Xinje XDPPro project, PLC1: XD5-60-6Pls (software 3.4 2016-10-12)

PROGRAM Ladder

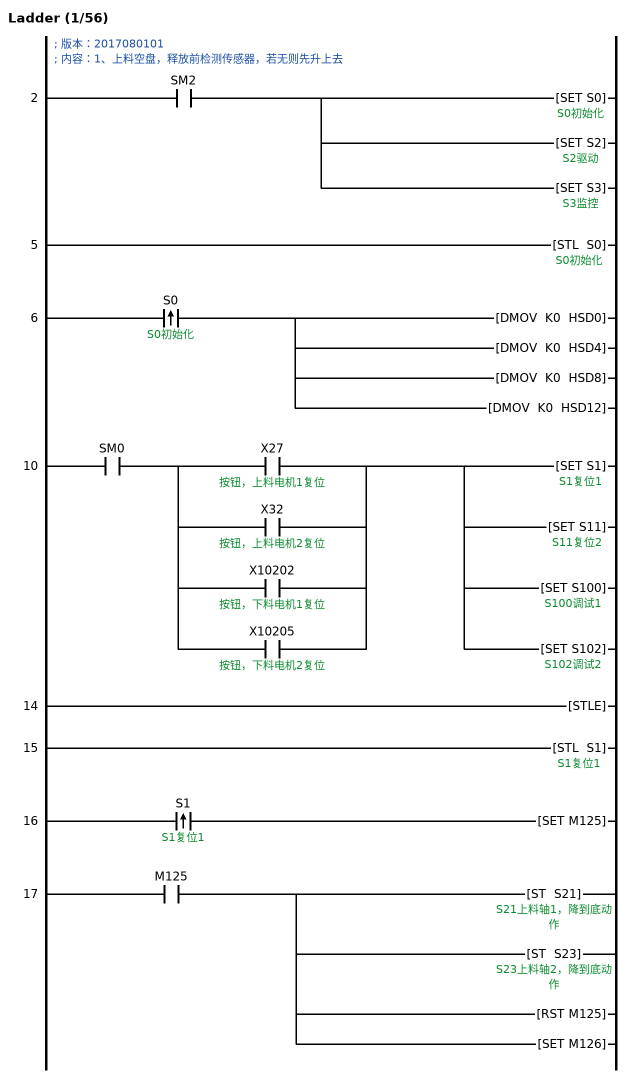
; 版本：2017080101
; 内容：1、上料空盘，释放前检测传感器，若无则先升上去
LD     SM2
SET    S0	; S0初始化
SET    S2	; S2驱动
SET    S3	; S3监控
STL    S0	; S0初始化
LDP    S0	; S0初始化
DMOV   K0 HSD0
DMOV   K0 HSD4
DMOV   K0 HSD8
DMOV   K0 HSD12
LD     SM0
LD     X27	; 按钮，上料电机1复位
OR     X32	; 按钮，上料电机2复位
OR     X10202	; 按钮，下料电机1复位
OR     X10205	; 按钮，下料电机2复位
ANB
SET    S1	; S1复位1
SET    S11	; S11复位2
SET    S100	; S100调试1
SET    S102	; S102调试2
STLE
STL    S1	; S1复位1
LDP    S1	; S1复位1
SET    M125
LD     M125
ST     S21	; S21上料轴1，降到底动作
ST     S23	; S23上料轴2，降到底动作
RST    M125
SET    M126

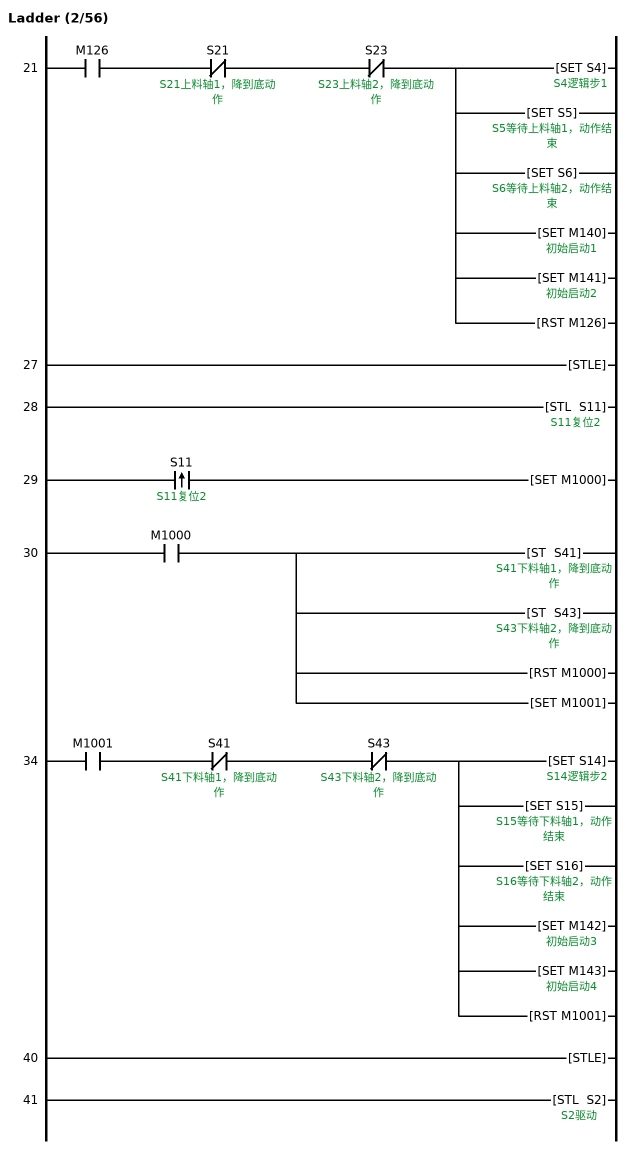
LD     M126
ANI    S21	; S21上料轴1，降到底动作
ANI    S23	; S23上料轴2，降到底动作
SET    S4	; S4逻辑步1
SET    S5	; S5等待上料轴1，动作结束
SET    S6	; S6等待上料轴2，动作结束
SET    M140	; 初始启动1
SET    M141	; 初始启动2
RST    M126
STLE
STL    S11	; S11复位2
LDP    S11	; S11复位2
SET    M1000
LD     M1000
ST     S41	; S41下料轴1，降到底动作
ST     S43	; S43下料轴2，降到底动作
RST    M1000
SET    M1001
LD     M1001
ANI    S41	; S41下料轴1，降到底动作
ANI    S43	; S43下料轴2，降到底动作
SET    S14	; S14逻辑步2
SET    S15	; S15等待下料轴1，动作结束
SET    S16	; S16等待下料轴2，动作结束
SET    M142	; 初始启动3
SET    M143	; 初始启动4
RST    M1001
STLE
STL    S2	; S2驱动

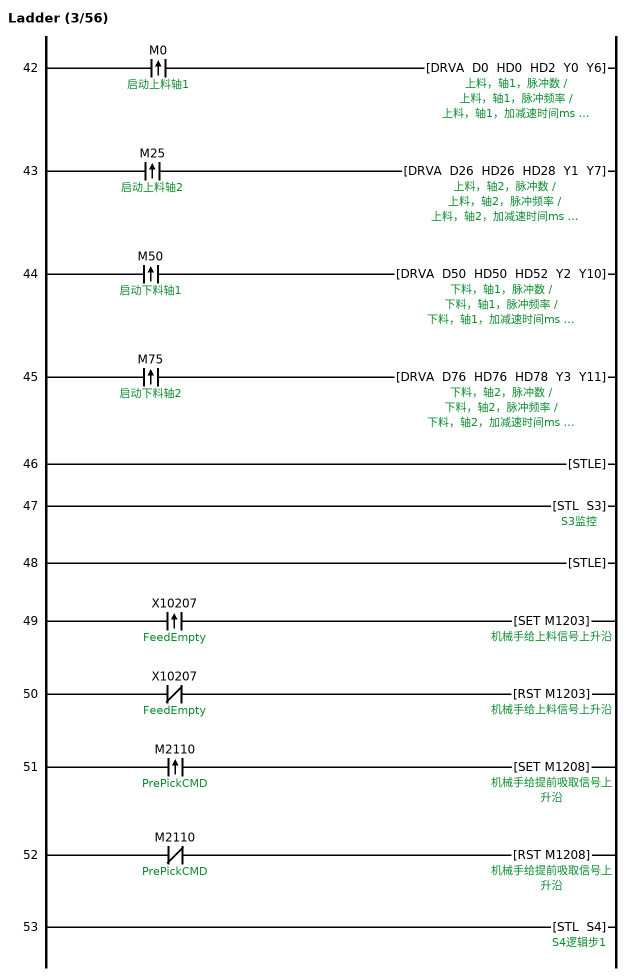
LDP    M0	; 启动上料轴1
DRVA   D0 HD0 HD2 Y0 Y6	; 上料，轴1，脉冲数 / 上料，轴1，脉冲频率 / 上料，轴1，加减速时间ms / 上料1电机脉冲 / 上料1电机方向
LDP    M25	; 启动上料轴2
DRVA   D26 HD26 HD28 Y1 Y7	; 上料，轴2，脉冲数 / 上料，轴2，脉冲频率 / 上料，轴2，加减速时间ms / 上料2电机脉冲 / 上料2电机方向
LDP    M50	; 启动下料轴1
DRVA   D50 HD50 HD52 Y2 Y10	; 下料，轴1，脉冲数 / 下料，轴1，脉冲频率 / 下料，轴1，加减速时间ms / 下料1电机脉冲 / 下料1电机方向
LDP    M75	; 启动下料轴2
DRVA   D76 HD76 HD78 Y3 Y11	; 下料，轴2，脉冲数 / 下料，轴2，脉冲频率 / 下料，轴2，加减速时间ms / 下料2电机脉冲 / 下料2电机方向
STLE
STL    S3	; S3监控
STLE
LDP    X10207	; FeedEmpty
SET    M1203	; 机械手给上料信号上升沿
LDI    X10207	; FeedEmpty
RST    M1203	; 机械手给上料信号上升沿
LDP    M2110	; PrePickCMD
SET    M1208	; 机械手给提前吸取信号上升沿
LDI    M2110	; PrePickCMD
RST    M1208	; 机械手给提前吸取信号上升沿
STL    S4	; S4逻辑步1

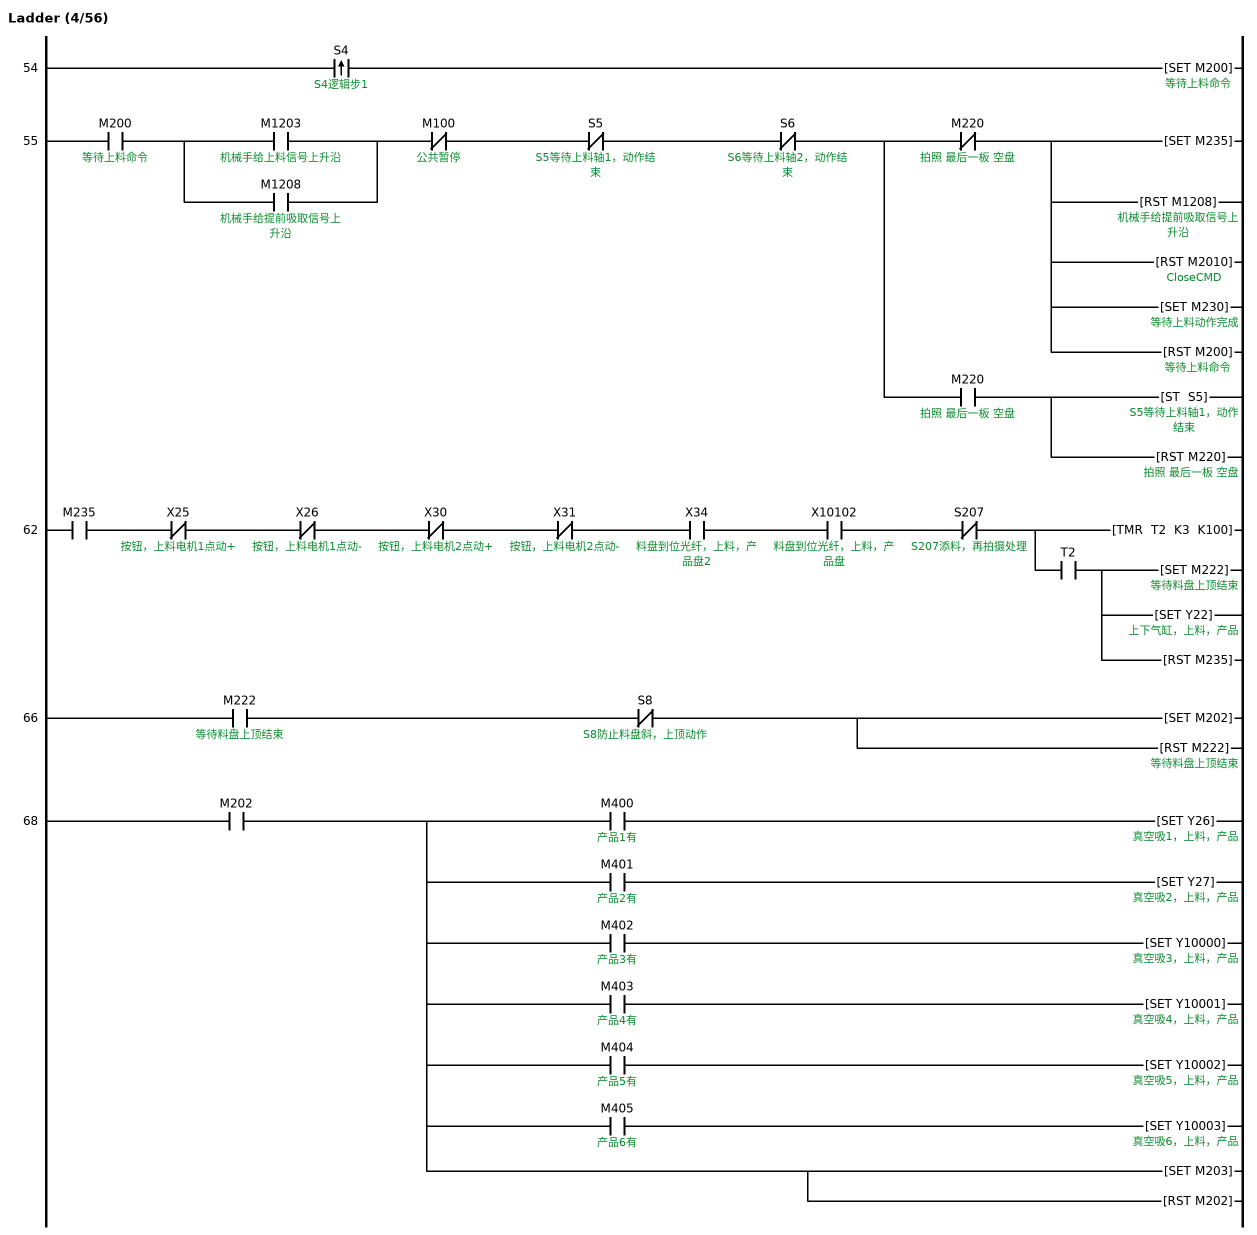
LDP    S4	; S4逻辑步1
SET    M200	; 等待上料命令
LD     M200	; 等待上料命令
LD     M1203	; 机械手给上料信号上升沿
OR     M1208	; 机械手给提前吸取信号上升沿
ANB
ANI    M100	; 公共暂停
ANI    S5	; S5等待上料轴1，动作结束
ANI    S6	; S6等待上料轴2，动作结束
MPS
ANI    M220	; 拍照 最后一板 空盘
SET    M235
RST    M1208	; 机械手给提前吸取信号上升沿
RST    M2010	; CloseCMD
SET    M230	; 等待上料动作完成
RST    M200	; 等待上料命令
MPP
AND    M220	; 拍照 最后一板 空盘
ST     S5	; S5等待上料轴1，动作结束
RST    M220	; 拍照 最后一板 空盘
LD     M235
ANI    X25	; 按钮，上料电机1点动+
ANI    X26	; 按钮，上料电机1点动-
ANI    X30	; 按钮，上料电机2点动+
ANI    X31	; 按钮，上料电机2点动-
AND    X34	; 料盘到位光纤，上料，产品盘2
AND    X10102	; 料盘到位光纤，上料，产品盘
ANI    S207	; S207添料，再拍摄处理
TMR    T2 K3 K100
AND    T2
SET    M222	; 等待料盘上顶结束
SET    Y22	; 上下气缸，上料，产品
RST    M235
LD     M222	; 等待料盘上顶结束
ANI    S8	; S8防止料盘斜，上顶动作
SET    M202
RST    M222	; 等待料盘上顶结束
LD     M202
MPS
AND    M400	; 产品1有
SET    Y26	; 真空吸1，上料，产品
MRD
AND    M401	; 产品2有
SET    Y27	; 真空吸2，上料，产品
MRD
AND    M402	; 产品3有
SET    Y10000	; 真空吸3，上料，产品
MRD
AND    M403	; 产品4有
SET    Y10001	; 真空吸4，上料，产品
MRD
AND    M404	; 产品5有
SET    Y10002	; 真空吸5，上料，产品
MRD
AND    M405	; 产品6有
SET    Y10003	; 真空吸6，上料，产品
MPP
SET    M203
RST    M202

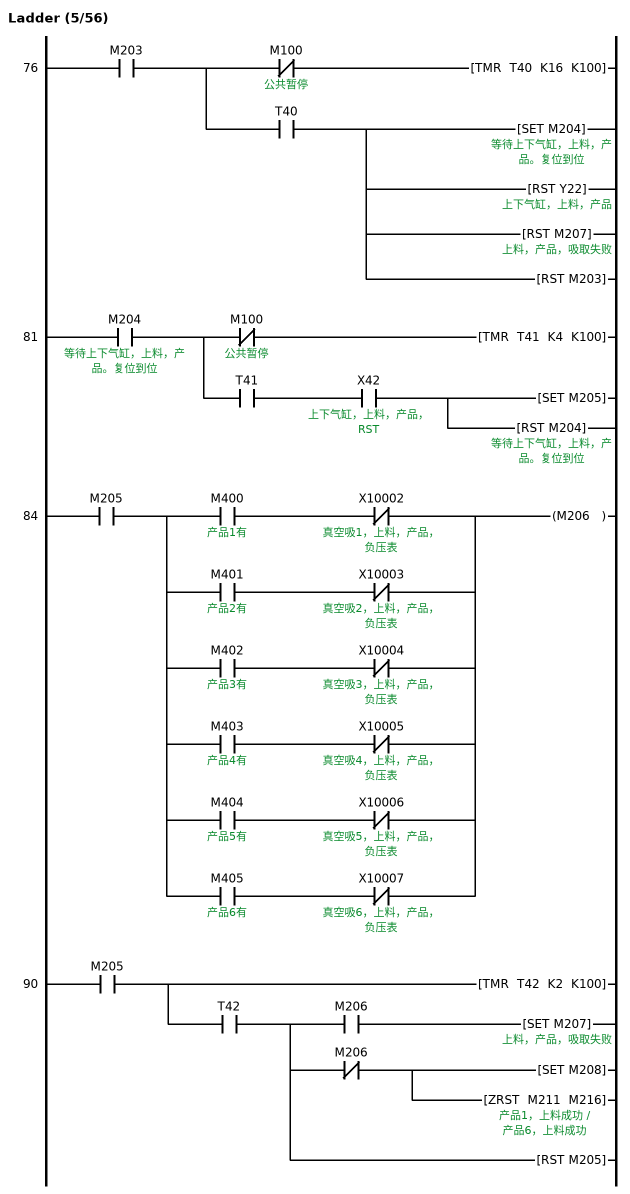
LD     M203
MPS
ANI    M100	; 公共暂停
TMR    T40 K16 K100
MPP
AND    T40
SET    M204	; 等待上下气缸，上料，产品。复位到位
RST    Y22	; 上下气缸，上料，产品
RST    M207	; 上料，产品，吸取失败
RST    M203
LD     M204	; 等待上下气缸，上料，产品。复位到位
MPS
ANI    M100	; 公共暂停
TMR    T41 K4 K100
MPP
AND    T41
AND    X42	; 上下气缸，上料，产品，RST
SET    M205
RST    M204	; 等待上下气缸，上料，产品。复位到位
LD     M205
LD     M400	; 产品1有
ANI    X10002	; 真空吸1，上料，产品，负压表
LD     M401	; 产品2有
ANI    X10003	; 真空吸2，上料，产品，负压表
ORB
LD     M402	; 产品3有
ANI    X10004	; 真空吸3，上料，产品，负压表
ORB
LD     M403	; 产品4有
ANI    X10005	; 真空吸4，上料，产品，负压表
ORB
LD     M404	; 产品5有
ANI    X10006	; 真空吸5，上料，产品，负压表
ORB
LD     M405	; 产品6有
ANI    X10007	; 真空吸6，上料，产品，负压表
ORB
ANB
OUT    M206
LD     M205
TMR    T42 K2 K100
AND    T42
MPS
AND    M206
SET    M207	; 上料，产品，吸取失败
MRD
ANI    M206
SET    M208
ZRST   M211 M216	; 产品1，上料成功 / 产品6，上料成功
MPP
RST    M205

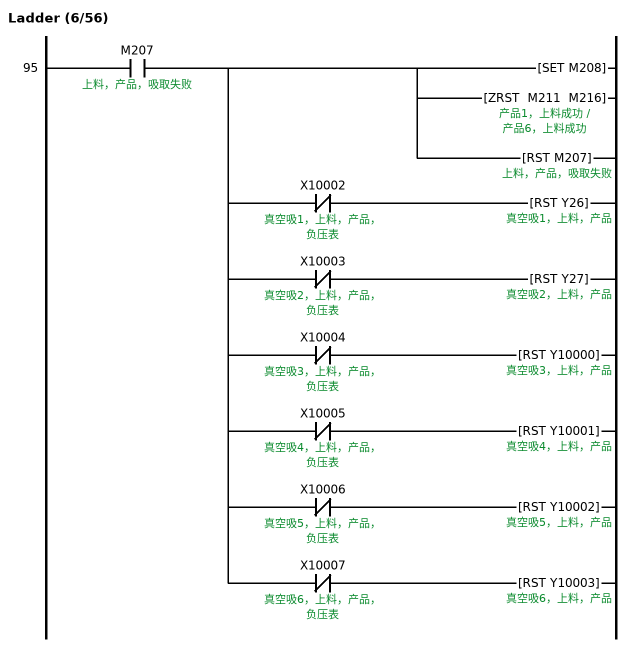
LD     M207	; 上料，产品，吸取失败
SET    M208
ZRST   M211 M216	; 产品1，上料成功 / 产品6，上料成功
RST    M207	; 上料，产品，吸取失败
MPS
ANI    X10002	; 真空吸1，上料，产品，负压表
RST    Y26	; 真空吸1，上料，产品
MRD
ANI    X10003	; 真空吸2，上料，产品，负压表
RST    Y27	; 真空吸2，上料，产品
MRD
ANI    X10004	; 真空吸3，上料，产品，负压表
RST    Y10000	; 真空吸3，上料，产品
MRD
ANI    X10005	; 真空吸4，上料，产品，负压表
RST    Y10001	; 真空吸4，上料，产品
MRD
ANI    X10006	; 真空吸5，上料，产品，负压表
RST    Y10002	; 真空吸5，上料，产品
MPP
ANI    X10007	; 真空吸6，上料，产品，负压表
RST    Y10003	; 真空吸6，上料，产品

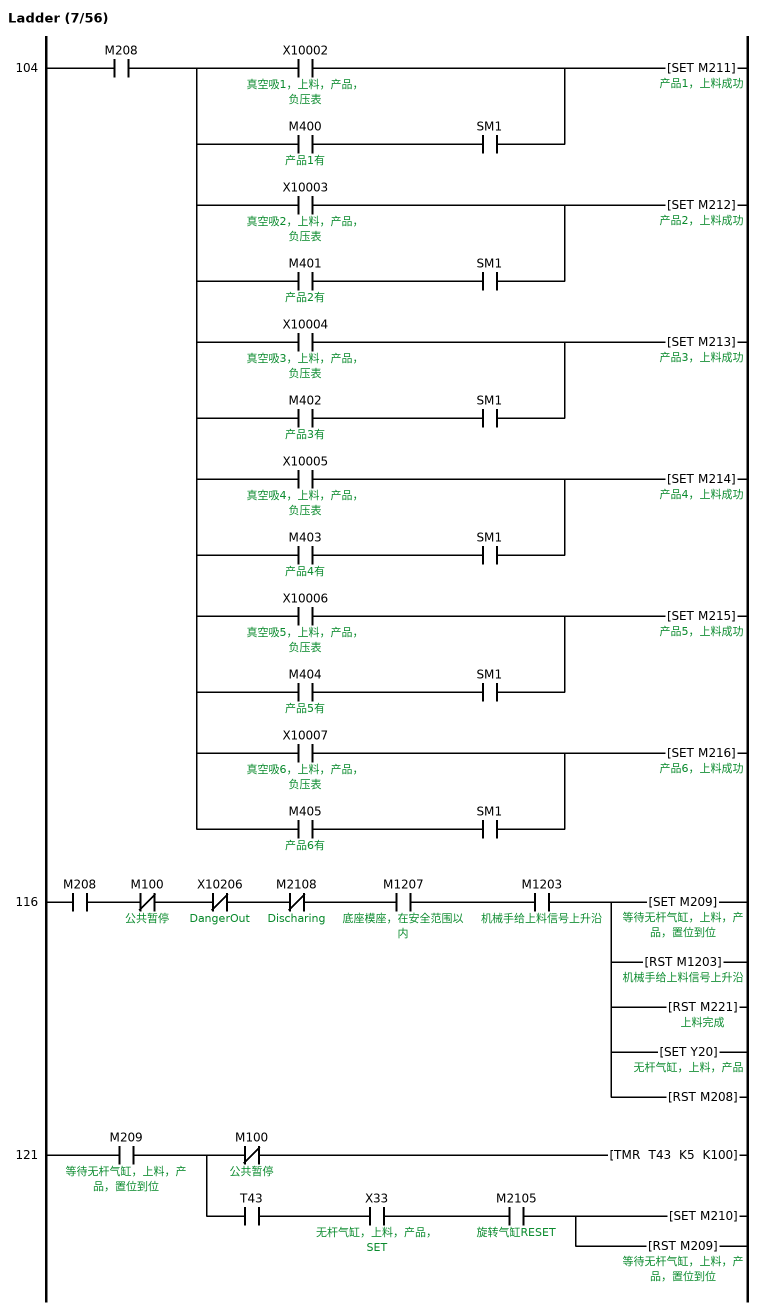
LD     M208
MPS
LD     X10002	; 真空吸1，上料，产品，负压表
LD     M400	; 产品1有
AND    SM1
ORB
ANB
SET    M211	; 产品1，上料成功
MRD
LD     X10003	; 真空吸2，上料，产品，负压表
LD     M401	; 产品2有
AND    SM1
ORB
ANB
SET    M212	; 产品2，上料成功
MRD
LD     X10004	; 真空吸3，上料，产品，负压表
LD     M402	; 产品3有
AND    SM1
ORB
ANB
SET    M213	; 产品3，上料成功
MRD
LD     X10005	; 真空吸4，上料，产品，负压表
LD     M403	; 产品4有
AND    SM1
ORB
ANB
SET    M214	; 产品4，上料成功
MRD
LD     X10006	; 真空吸5，上料，产品，负压表
LD     M404	; 产品5有
AND    SM1
ORB
ANB
SET    M215	; 产品5，上料成功
MPP
LD     X10007	; 真空吸6，上料，产品，负压表
LD     M405	; 产品6有
AND    SM1
ORB
ANB
SET    M216	; 产品6，上料成功
LD     M208
ANI    M100	; 公共暂停
ANI    X10206	; DangerOut
ANI    M2108	; Discharing
AND    M1207	; 底座模座，在安全范围以内
AND    M1203	; 机械手给上料信号上升沿
SET    M209	; 等待无杆气缸，上料，产品，置位到位
RST    M1203	; 机械手给上料信号上升沿
RST    M221	; 上料完成
SET    Y20	; 无杆气缸，上料，产品
RST    M208
LD     M209	; 等待无杆气缸，上料，产品，置位到位
MPS
ANI    M100	; 公共暂停
TMR    T43 K5 K100
MPP
AND    T43
AND    X33	; 无杆气缸，上料，产品，SET
AND    M2105	; 旋转气缸RESET
SET    M210
RST    M209	; 等待无杆气缸，上料，产品，置位到位

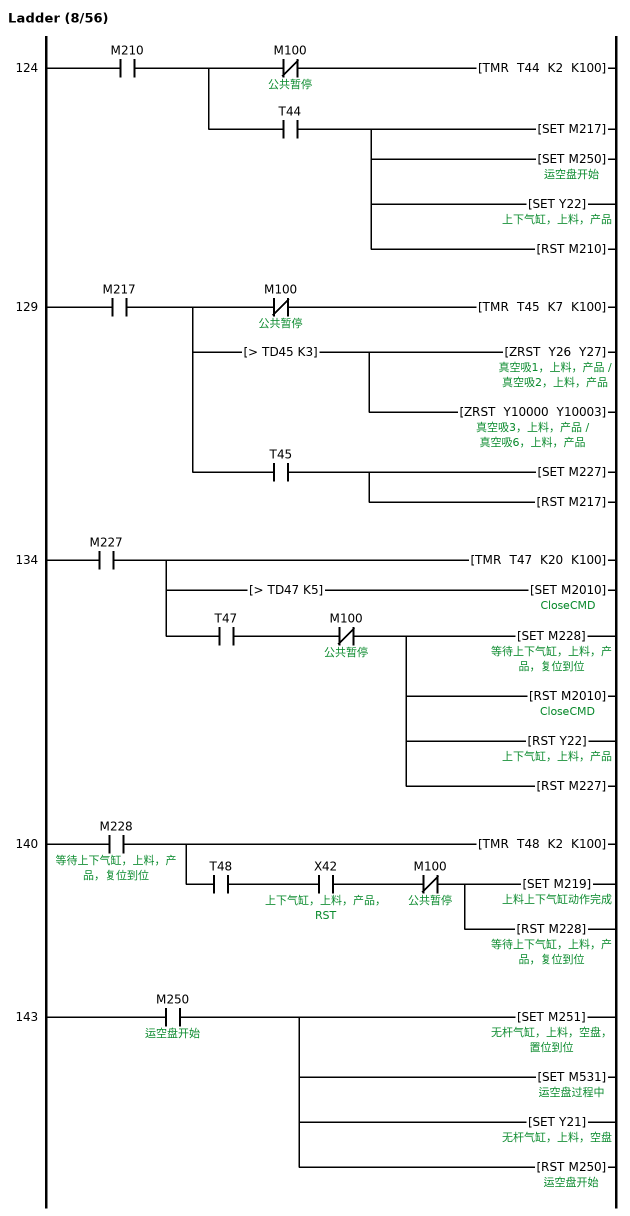
LD     M210
MPS
ANI    M100	; 公共暂停
TMR    T44 K2 K100
MPP
AND    T44
SET    M217
SET    M250	; 运空盘开始
SET    Y22	; 上下气缸，上料，产品
RST    M210
LD     M217
MPS
ANI    M100	; 公共暂停
TMR    T45 K7 K100
MRD
AND>   TD45 K3
ZRST   Y26 Y27	; 真空吸1，上料，产品 / 真空吸2，上料，产品
ZRST   Y10000 Y10003	; 真空吸3，上料，产品 / 真空吸6，上料，产品
MPP
AND    T45
SET    M227
RST    M217
LD     M227
TMR    T47 K20 K100
MPS
AND>   TD47 K5
SET    M2010	; CloseCMD
MPP
AND    T47
ANI    M100	; 公共暂停
SET    M228	; 等待上下气缸，上料，产品，复位到位
RST    M2010	; CloseCMD
RST    Y22	; 上下气缸，上料，产品
RST    M227
LD     M228	; 等待上下气缸，上料，产品，复位到位
TMR    T48 K2 K100
AND    T48
AND    X42	; 上下气缸，上料，产品，RST
ANI    M100	; 公共暂停
SET    M219	; 上料上下气缸动作完成
RST    M228	; 等待上下气缸，上料，产品，复位到位
LD     M250	; 运空盘开始
SET    M251	; 无杆气缸，上料，空盘，置位到位
SET    M531	; 运空盘过程中
SET    Y21	; 无杆气缸，上料，空盘
RST    M250	; 运空盘开始

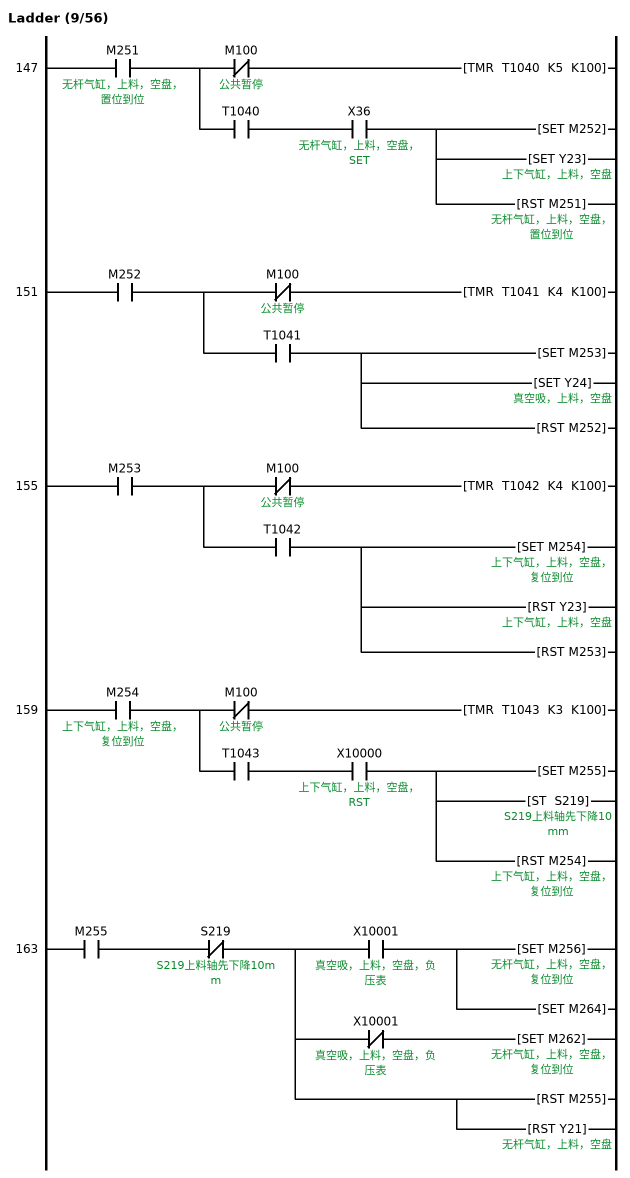
LD     M251	; 无杆气缸，上料，空盘，置位到位
MPS
ANI    M100	; 公共暂停
TMR    T1040 K5 K100
MPP
AND    T1040
AND    X36	; 无杆气缸，上料，空盘，SET
SET    M252
SET    Y23	; 上下气缸，上料，空盘
RST    M251	; 无杆气缸，上料，空盘，置位到位
LD     M252
MPS
ANI    M100	; 公共暂停
TMR    T1041 K4 K100
MPP
AND    T1041
SET    M253
SET    Y24	; 真空吸，上料，空盘
RST    M252
LD     M253
MPS
ANI    M100	; 公共暂停
TMR    T1042 K4 K100
MPP
AND    T1042
SET    M254	; 上下气缸，上料，空盘，复位到位
RST    Y23	; 上下气缸，上料，空盘
RST    M253
LD     M254	; 上下气缸，上料，空盘，复位到位
MPS
ANI    M100	; 公共暂停
TMR    T1043 K3 K100
MPP
AND    T1043
AND    X10000	; 上下气缸，上料，空盘，RST
SET    M255
ST     S219	; S219上料轴先下降10mm
RST    M254	; 上下气缸，上料，空盘，复位到位
LD     M255
ANI    S219	; S219上料轴先下降10mm
MPS
AND    X10001	; 真空吸，上料，空盘，负压表
SET    M256	; 无杆气缸，上料，空盘，复位到位
SET    M264
MRD
ANI    X10001	; 真空吸，上料，空盘，负压表
SET    M262	; 无杆气缸，上料，空盘，复位到位
MPP
RST    M255
RST    Y21	; 无杆气缸，上料，空盘

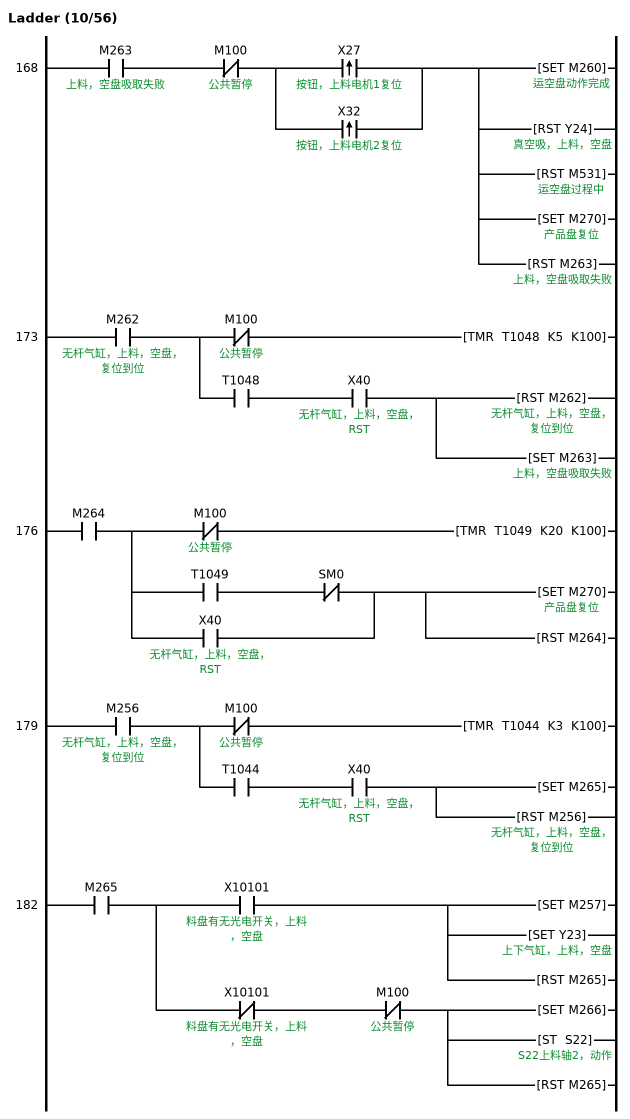
LD     M263	; 上料，空盘吸取失败
ANI    M100	; 公共暂停
LDP    X27	; 按钮，上料电机1复位
ORP    X32	; 按钮，上料电机2复位
ANB
SET    M260	; 运空盘动作完成
RST    Y24	; 真空吸，上料，空盘
RST    M531	; 运空盘过程中
SET    M270	; 产品盘复位
RST    M263	; 上料，空盘吸取失败
LD     M262	; 无杆气缸，上料，空盘，复位到位
MPS
ANI    M100	; 公共暂停
TMR    T1048 K5 K100
MPP
AND    T1048
AND    X40	; 无杆气缸，上料，空盘，RST
RST    M262	; 无杆气缸，上料，空盘，复位到位
SET    M263	; 上料，空盘吸取失败
LD     M264
MPS
ANI    M100	; 公共暂停
TMR    T1049 K20 K100
MPP
LD     T1049
ANI    SM0
OR     X40	; 无杆气缸，上料，空盘，RST
ANB
SET    M270	; 产品盘复位
RST    M264
LD     M256	; 无杆气缸，上料，空盘，复位到位
MPS
ANI    M100	; 公共暂停
TMR    T1044 K3 K100
MPP
AND    T1044
AND    X40	; 无杆气缸，上料，空盘，RST
SET    M265
RST    M256	; 无杆气缸，上料，空盘，复位到位
LD     M265
MPS
AND    X10101	; 料盘有无光电开关，上料，空盘
SET    M257
SET    Y23	; 上下气缸，上料，空盘
RST    M265
MPP
ANI    X10101	; 料盘有无光电开关，上料，空盘
ANI    M100	; 公共暂停
SET    M266
ST     S22	; S22上料轴2，动作
RST    M265

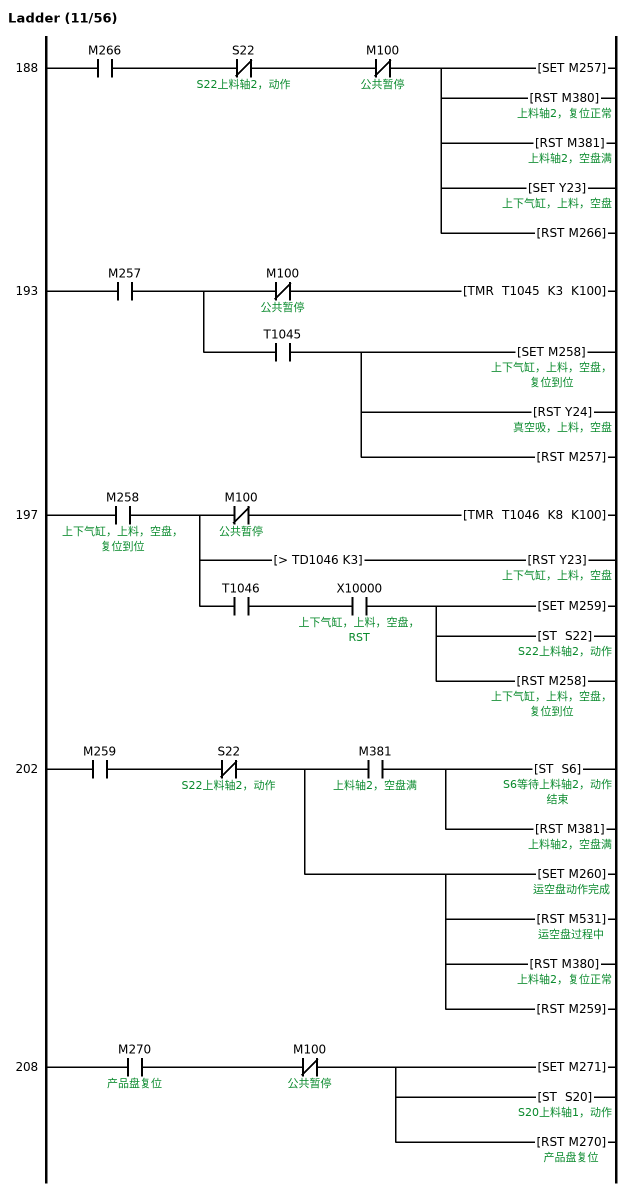
LD     M266
ANI    S22	; S22上料轴2，动作
ANI    M100	; 公共暂停
SET    M257
RST    M380	; 上料轴2，复位正常
RST    M381	; 上料轴2，空盘满
SET    Y23	; 上下气缸，上料，空盘
RST    M266
LD     M257
MPS
ANI    M100	; 公共暂停
TMR    T1045 K3 K100
MPP
AND    T1045
SET    M258	; 上下气缸，上料，空盘，复位到位
RST    Y24	; 真空吸，上料，空盘
RST    M257
LD     M258	; 上下气缸，上料，空盘，复位到位
MPS
ANI    M100	; 公共暂停
TMR    T1046 K8 K100
MRD
AND>   TD1046 K3
RST    Y23	; 上下气缸，上料，空盘
MPP
AND    T1046
AND    X10000	; 上下气缸，上料，空盘，RST
SET    M259
ST     S22	; S22上料轴2，动作
RST    M258	; 上下气缸，上料，空盘，复位到位
LD     M259
ANI    S22	; S22上料轴2，动作
MPS
AND    M381	; 上料轴2，空盘满
ST     S6	; S6等待上料轴2，动作结束
RST    M381	; 上料轴2，空盘满
MPP
SET    M260	; 运空盘动作完成
RST    M531	; 运空盘过程中
RST    M380	; 上料轴2，复位正常
RST    M259
LD     M270	; 产品盘复位
ANI    M100	; 公共暂停
SET    M271
ST     S20	; S20上料轴1，动作
RST    M270	; 产品盘复位

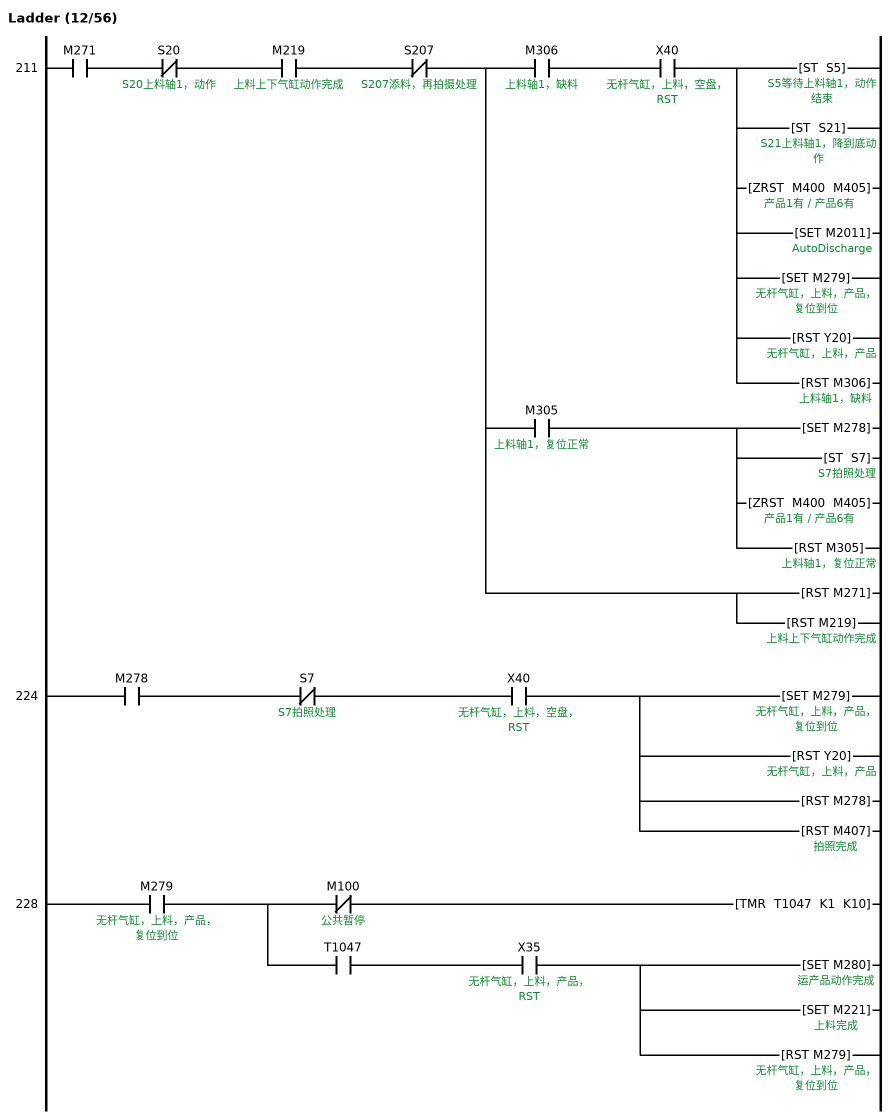
LD     M271
ANI    S20	; S20上料轴1，动作
AND    M219	; 上料上下气缸动作完成
ANI    S207	; S207添料，再拍摄处理
MPS
AND    M306	; 上料轴1，缺料
AND    X40	; 无杆气缸，上料，空盘，RST
ST     S5	; S5等待上料轴1，动作结束
ST     S21	; S21上料轴1，降到底动作
ZRST   M400 M405	; 产品1有 / 产品6有
SET    M2011	; AutoDischarge
SET    M279	; 无杆气缸，上料，产品，复位到位
RST    Y20	; 无杆气缸，上料，产品
RST    M306	; 上料轴1，缺料
MRD
AND    M305	; 上料轴1，复位正常
SET    M278
ST     S7	; S7拍照处理
ZRST   M400 M405	; 产品1有 / 产品6有
RST    M305	; 上料轴1，复位正常
MPP
RST    M271
RST    M219	; 上料上下气缸动作完成
LD     M278
ANI    S7	; S7拍照处理
AND    X40	; 无杆气缸，上料，空盘，RST
SET    M279	; 无杆气缸，上料，产品，复位到位
RST    Y20	; 无杆气缸，上料，产品
RST    M278
RST    M407	; 拍照完成
LD     M279	; 无杆气缸，上料，产品，复位到位
MPS
ANI    M100	; 公共暂停
TMR    T1047 K1 K10
MPP
AND    T1047
AND    X35	; 无杆气缸，上料，产品，RST
SET    M280	; 运产品动作完成
SET    M221	; 上料完成
RST    M279	; 无杆气缸，上料，产品，复位到位

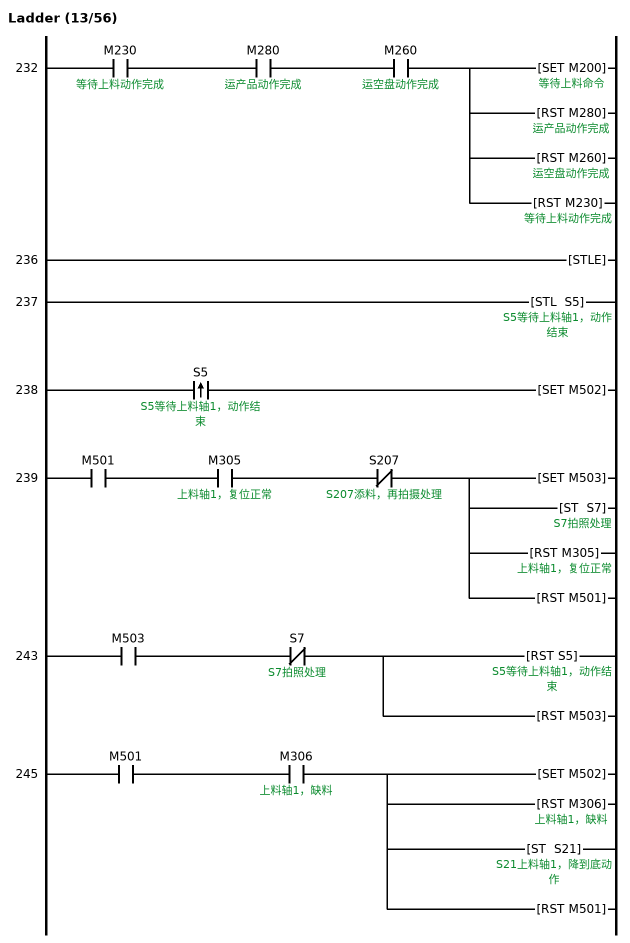
LD     M230	; 等待上料动作完成
AND    M280	; 运产品动作完成
AND    M260	; 运空盘动作完成
SET    M200	; 等待上料命令
RST    M280	; 运产品动作完成
RST    M260	; 运空盘动作完成
RST    M230	; 等待上料动作完成
STLE
STL    S5	; S5等待上料轴1，动作结束
LDP    S5	; S5等待上料轴1，动作结束
SET    M502
LD     M501
AND    M305	; 上料轴1，复位正常
ANI    S207	; S207添料，再拍摄处理
SET    M503
ST     S7	; S7拍照处理
RST    M305	; 上料轴1，复位正常
RST    M501
LD     M503
ANI    S7	; S7拍照处理
RST    S5	; S5等待上料轴1，动作结束
RST    M503
LD     M501
AND    M306	; 上料轴1，缺料
SET    M502
RST    M306	; 上料轴1，缺料
ST     S21	; S21上料轴1，降到底动作
RST    M501

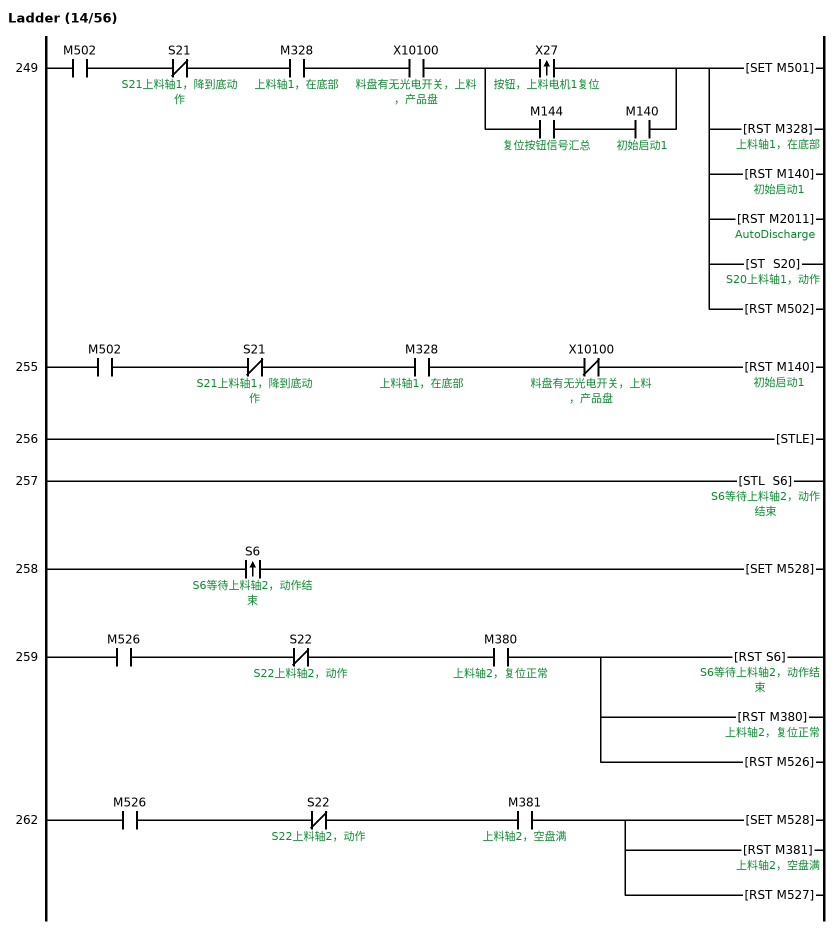
LD     M502
ANI    S21	; S21上料轴1，降到底动作
AND    M328	; 上料轴1，在底部
AND    X10100	; 料盘有无光电开关，上料，产品盘
LDP    X27	; 按钮，上料电机1复位
LD     M144	; 复位按钮信号汇总
AND    M140	; 初始启动1
ORB
ANB
SET    M501
RST    M328	; 上料轴1，在底部
RST    M140	; 初始启动1
RST    M2011	; AutoDischarge
ST     S20	; S20上料轴1，动作
RST    M502
LD     M502
ANI    S21	; S21上料轴1，降到底动作
AND    M328	; 上料轴1，在底部
ANI    X10100	; 料盘有无光电开关，上料，产品盘
RST    M140	; 初始启动1
STLE
STL    S6	; S6等待上料轴2，动作结束
LDP    S6	; S6等待上料轴2，动作结束
SET    M528
LD     M526
ANI    S22	; S22上料轴2，动作
AND    M380	; 上料轴2，复位正常
RST    S6	; S6等待上料轴2，动作结束
RST    M380	; 上料轴2，复位正常
RST    M526
LD     M526
ANI    S22	; S22上料轴2，动作
AND    M381	; 上料轴2，空盘满
SET    M528
RST    M381	; 上料轴2，空盘满
RST    M527

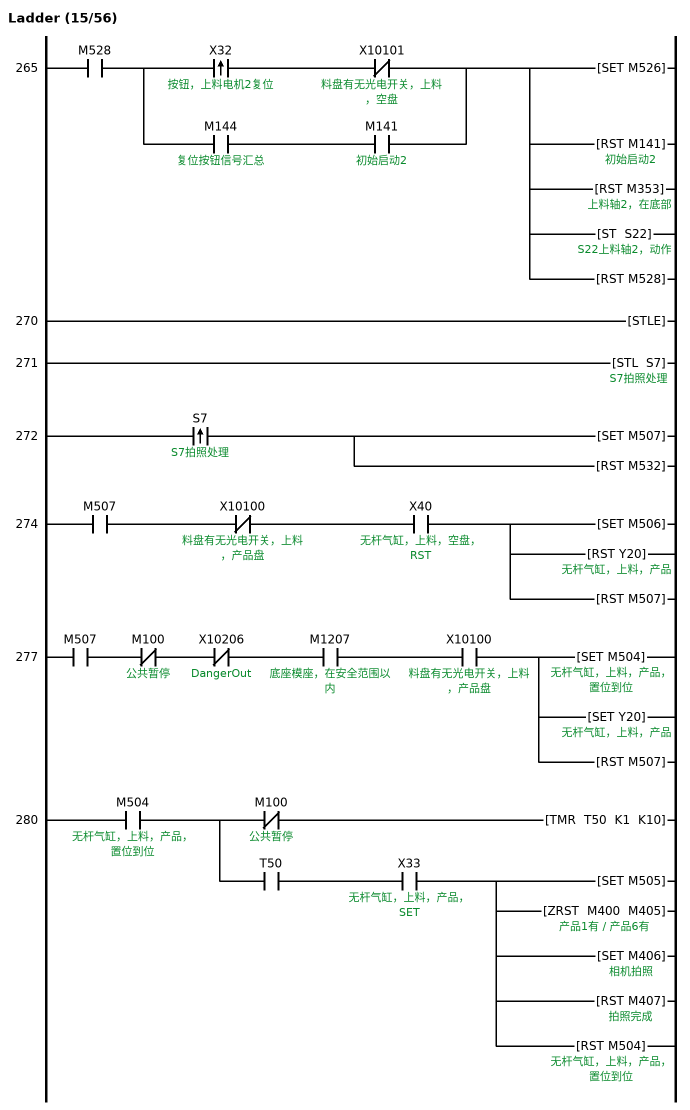
LD     M528
LDP    X32	; 按钮，上料电机2复位
ANI    X10101	; 料盘有无光电开关，上料，空盘
LD     M144	; 复位按钮信号汇总
AND    M141	; 初始启动2
ORB
ANB
SET    M526
RST    M141	; 初始启动2
RST    M353	; 上料轴2，在底部
ST     S22	; S22上料轴2，动作
RST    M528
STLE
STL    S7	; S7拍照处理
LDP    S7	; S7拍照处理
SET    M507
RST    M532
LD     M507
ANI    X10100	; 料盘有无光电开关，上料，产品盘
AND    X40	; 无杆气缸，上料，空盘，RST
SET    M506
RST    Y20	; 无杆气缸，上料，产品
RST    M507
LD     M507
ANI    M100	; 公共暂停
ANI    X10206	; DangerOut
AND    M1207	; 底座模座，在安全范围以内
AND    X10100	; 料盘有无光电开关，上料，产品盘
SET    M504	; 无杆气缸，上料，产品，置位到位
SET    Y20	; 无杆气缸，上料，产品
RST    M507
LD     M504	; 无杆气缸，上料，产品，置位到位
MPS
ANI    M100	; 公共暂停
TMR    T50 K1 K10
MPP
AND    T50
AND    X33	; 无杆气缸，上料，产品，SET
SET    M505
ZRST   M400 M405	; 产品1有 / 产品6有
SET    M406	; 相机拍照
RST    M407	; 拍照完成
RST    M504	; 无杆气缸，上料，产品，置位到位

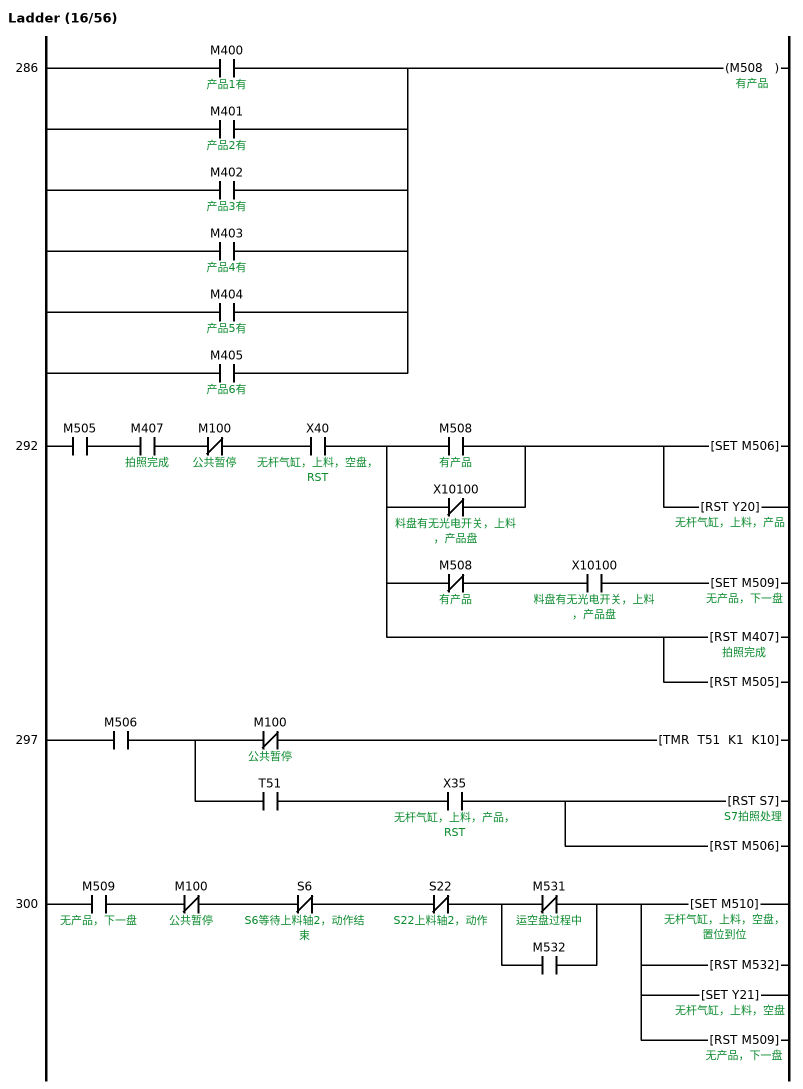
LD     M400	; 产品1有
OR     M401	; 产品2有
OR     M402	; 产品3有
OR     M403	; 产品4有
OR     M404	; 产品5有
OR     M405	; 产品6有
OUT    M508	; 有产品
LD     M505
AND    M407	; 拍照完成
ANI    M100	; 公共暂停
AND    X40	; 无杆气缸，上料，空盘，RST
MPS
LD     M508	; 有产品
ORI    X10100	; 料盘有无光电开关，上料，产品盘
ANB
SET    M506
RST    Y20	; 无杆气缸，上料，产品
MRD
ANI    M508	; 有产品
AND    X10100	; 料盘有无光电开关，上料，产品盘
SET    M509	; 无产品，下一盘
MPP
RST    M407	; 拍照完成
RST    M505
LD     M506
MPS
ANI    M100	; 公共暂停
TMR    T51 K1 K10
MPP
AND    T51
AND    X35	; 无杆气缸，上料，产品，RST
RST    S7	; S7拍照处理
RST    M506
LD     M509	; 无产品，下一盘
ANI    M100	; 公共暂停
ANI    S6	; S6等待上料轴2，动作结束
ANI    S22	; S22上料轴2，动作
LDI    M531	; 运空盘过程中
OR     M532
ANB
SET    M510	; 无杆气缸，上料，空盘，置位到位
RST    M532
SET    Y21	; 无杆气缸，上料，空盘
RST    M509	; 无产品，下一盘

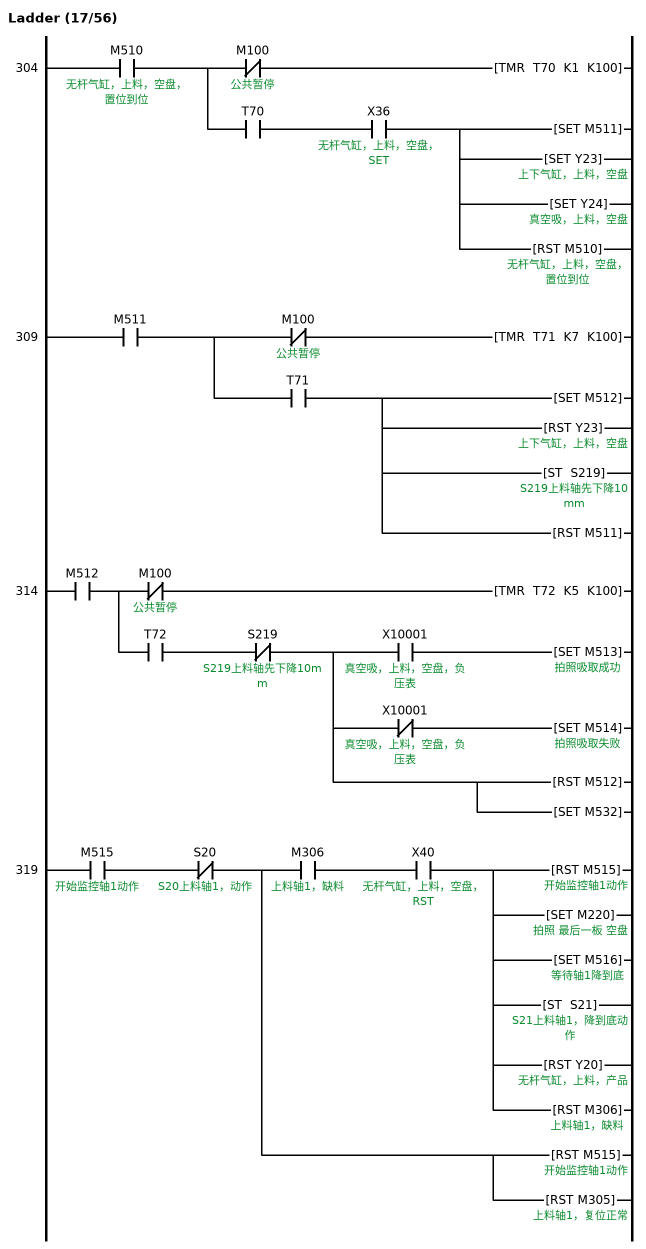
LD     M510	; 无杆气缸，上料，空盘，置位到位
MPS
ANI    M100	; 公共暂停
TMR    T70 K1 K100
MPP
AND    T70
AND    X36	; 无杆气缸，上料，空盘，SET
SET    M511
SET    Y23	; 上下气缸，上料，空盘
SET    Y24	; 真空吸，上料，空盘
RST    M510	; 无杆气缸，上料，空盘，置位到位
LD     M511
MPS
ANI    M100	; 公共暂停
TMR    T71 K7 K100
MPP
AND    T71
SET    M512
RST    Y23	; 上下气缸，上料，空盘
ST     S219	; S219上料轴先下降10mm
RST    M511
LD     M512
MPS
ANI    M100	; 公共暂停
TMR    T72 K5 K100
MPP
AND    T72
ANI    S219	; S219上料轴先下降10mm
MPS
AND    X10001	; 真空吸，上料，空盘，负压表
SET    M513	; 拍照吸取成功
MRD
ANI    X10001	; 真空吸，上料，空盘，负压表
SET    M514	; 拍照吸取失败
MPP
RST    M512
SET    M532
LD     M515	; 开始监控轴1动作
ANI    S20	; S20上料轴1，动作
MPS
AND    M306	; 上料轴1，缺料
AND    X40	; 无杆气缸，上料，空盘，RST
RST    M515	; 开始监控轴1动作
SET    M220	; 拍照 最后一板 空盘
SET    M516	; 等待轴1降到底
ST     S21	; S21上料轴1，降到底动作
RST    Y20	; 无杆气缸，上料，产品
RST    M306	; 上料轴1，缺料
MPP
RST    M515	; 开始监控轴1动作
RST    M305	; 上料轴1，复位正常

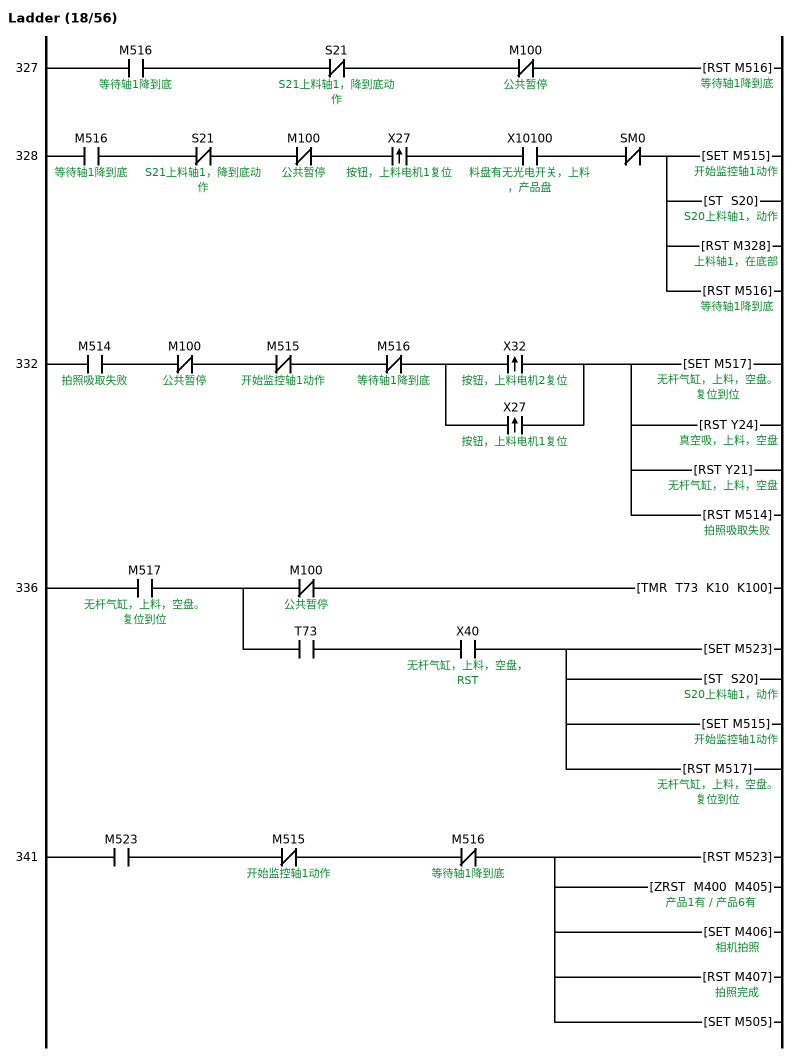
LD     M516	; 等待轴1降到底
ANI    S21	; S21上料轴1，降到底动作
ANI    M100	; 公共暂停
RST    M516	; 等待轴1降到底
LD     M516	; 等待轴1降到底
ANI    S21	; S21上料轴1，降到底动作
ANI    M100	; 公共暂停
ANDP   X27	; 按钮，上料电机1复位
AND    X10100	; 料盘有无光电开关，上料，产品盘
ANI    SM0
SET    M515	; 开始监控轴1动作
ST     S20	; S20上料轴1，动作
RST    M328	; 上料轴1，在底部
RST    M516	; 等待轴1降到底
LD     M514	; 拍照吸取失败
ANI    M100	; 公共暂停
ANI    M515	; 开始监控轴1动作
ANI    M516	; 等待轴1降到底
LDP    X32	; 按钮，上料电机2复位
ORP    X27	; 按钮，上料电机1复位
ANB
SET    M517	; 无杆气缸，上料，空盘。复位到位
RST    Y24	; 真空吸，上料，空盘
RST    Y21	; 无杆气缸，上料，空盘
RST    M514	; 拍照吸取失败
LD     M517	; 无杆气缸，上料，空盘。复位到位
MPS
ANI    M100	; 公共暂停
TMR    T73 K10 K100
MPP
AND    T73
AND    X40	; 无杆气缸，上料，空盘，RST
SET    M523
ST     S20	; S20上料轴1，动作
SET    M515	; 开始监控轴1动作
RST    M517	; 无杆气缸，上料，空盘。复位到位
LD     M523
ANI    M515	; 开始监控轴1动作
ANI    M516	; 等待轴1降到底
RST    M523
ZRST   M400 M405	; 产品1有 / 产品6有
SET    M406	; 相机拍照
RST    M407	; 拍照完成
SET    M505

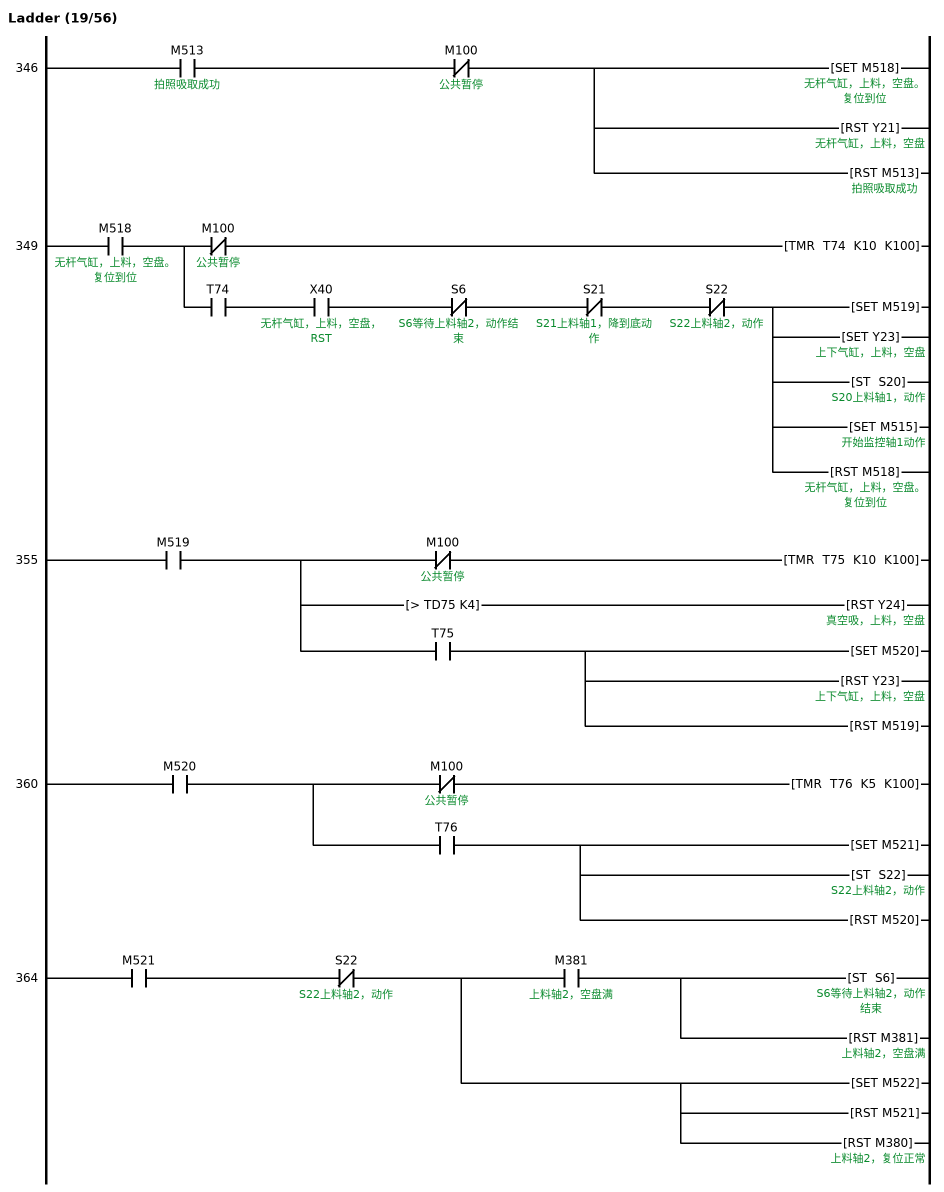
LD     M513	; 拍照吸取成功
ANI    M100	; 公共暂停
SET    M518	; 无杆气缸，上料，空盘。复位到位
RST    Y21	; 无杆气缸，上料，空盘
RST    M513	; 拍照吸取成功
LD     M518	; 无杆气缸，上料，空盘。复位到位
MPS
ANI    M100	; 公共暂停
TMR    T74 K10 K100
MPP
AND    T74
AND    X40	; 无杆气缸，上料，空盘，RST
ANI    S6	; S6等待上料轴2，动作结束
ANI    S21	; S21上料轴1，降到底动作
ANI    S22	; S22上料轴2，动作
SET    M519
SET    Y23	; 上下气缸，上料，空盘
ST     S20	; S20上料轴1，动作
SET    M515	; 开始监控轴1动作
RST    M518	; 无杆气缸，上料，空盘。复位到位
LD     M519
MPS
ANI    M100	; 公共暂停
TMR    T75 K10 K100
MRD
AND>   TD75 K4
RST    Y24	; 真空吸，上料，空盘
MPP
AND    T75
SET    M520
RST    Y23	; 上下气缸，上料，空盘
RST    M519
LD     M520
MPS
ANI    M100	; 公共暂停
TMR    T76 K5 K100
MPP
AND    T76
SET    M521
ST     S22	; S22上料轴2，动作
RST    M520
LD     M521
ANI    S22	; S22上料轴2，动作
MPS
AND    M381	; 上料轴2，空盘满
ST     S6	; S6等待上料轴2，动作结束
RST    M381	; 上料轴2，空盘满
MPP
SET    M522
RST    M521
RST    M380	; 上料轴2，复位正常

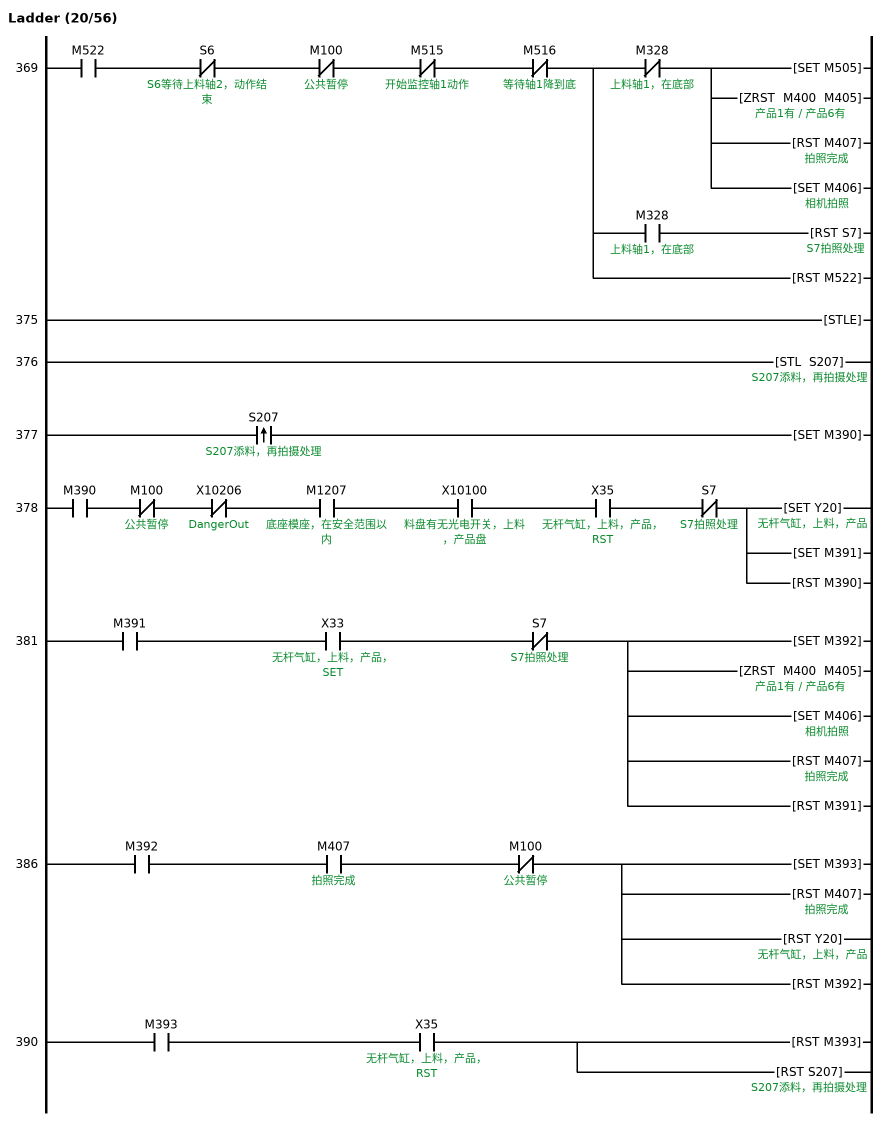
LD     M522
ANI    S6	; S6等待上料轴2，动作结束
ANI    M100	; 公共暂停
ANI    M515	; 开始监控轴1动作
ANI    M516	; 等待轴1降到底
MPS
ANI    M328	; 上料轴1，在底部
SET    M505
ZRST   M400 M405	; 产品1有 / 产品6有
RST    M407	; 拍照完成
SET    M406	; 相机拍照
MRD
AND    M328	; 上料轴1，在底部
RST    S7	; S7拍照处理
MPP
RST    M522
STLE
STL    S207	; S207添料，再拍摄处理
LDP    S207	; S207添料，再拍摄处理
SET    M390
LD     M390
ANI    M100	; 公共暂停
ANI    X10206	; DangerOut
AND    M1207	; 底座模座，在安全范围以内
AND    X10100	; 料盘有无光电开关，上料，产品盘
AND    X35	; 无杆气缸，上料，产品，RST
ANI    S7	; S7拍照处理
SET    Y20	; 无杆气缸，上料，产品
SET    M391
RST    M390
LD     M391
AND    X33	; 无杆气缸，上料，产品，SET
ANI    S7	; S7拍照处理
SET    M392
ZRST   M400 M405	; 产品1有 / 产品6有
SET    M406	; 相机拍照
RST    M407	; 拍照完成
RST    M391
LD     M392
AND    M407	; 拍照完成
ANI    M100	; 公共暂停
SET    M393
RST    M407	; 拍照完成
RST    Y20	; 无杆气缸，上料，产品
RST    M392
LD     M393
AND    X35	; 无杆气缸，上料，产品，RST
RST    M393
RST    S207	; S207添料，再拍摄处理

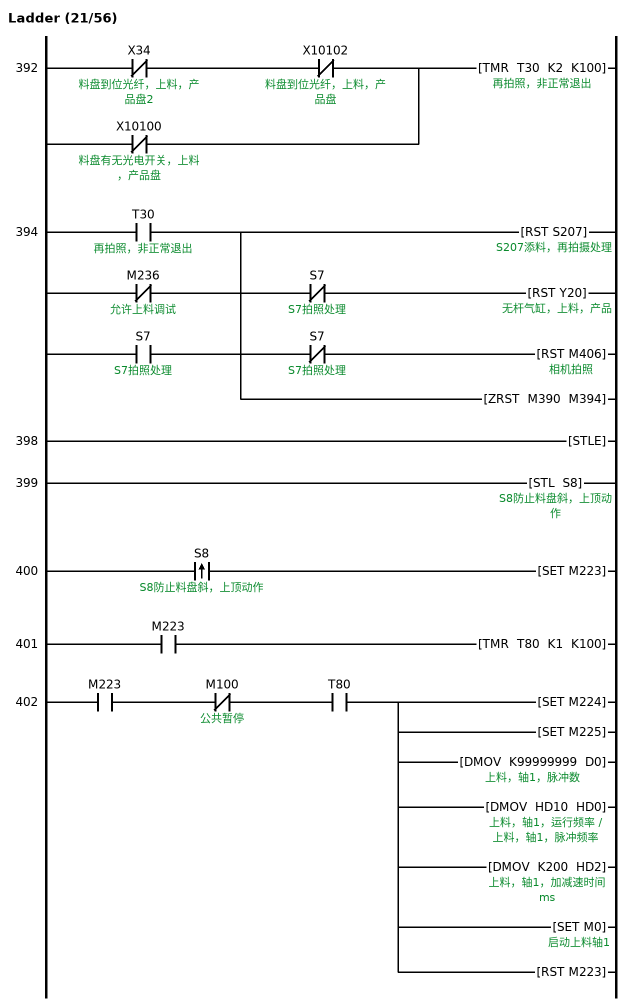
LDI    X34	; 料盘到位光纤，上料，产品盘2
ANI    X10102	; 料盘到位光纤，上料，产品盘
ORI    X10100	; 料盘有无光电开关，上料，产品盘
TMR    T30 K2 K100	; 再拍照，非正常退出
LD     T30	; 再拍照，非正常退出
ORI    M236	; 允许上料调试
OR     S7	; S7拍照处理
RST    S207	; S207添料，再拍摄处理
MPS
ANI    S7	; S7拍照处理
RST    Y20	; 无杆气缸，上料，产品
MRD
ANI    S7	; S7拍照处理
RST    M406	; 相机拍照
MPP
ZRST   M390 M394
STLE
STL    S8	; S8防止料盘斜，上顶动作
LDP    S8	; S8防止料盘斜，上顶动作
SET    M223
LD     M223
TMR    T80 K1 K100
LD     M223
ANI    M100	; 公共暂停
AND    T80
SET    M224
SET    M225
DMOV   K99999999 D0	; 上料，轴1，脉冲数
DMOV   HD10 HD0	; 上料，轴1，运行频率 / 上料，轴1，脉冲频率
DMOV   K200 HD2	; 上料，轴1，加减速时间ms
SET    M0	; 启动上料轴1
RST    M223

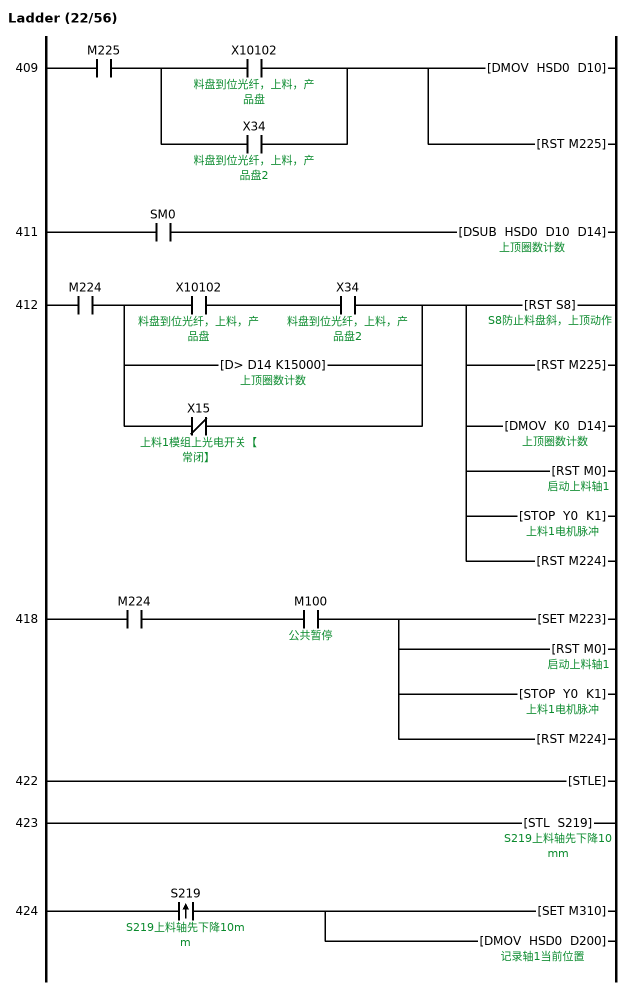
LD     M225
LD     X10102	; 料盘到位光纤，上料，产品盘
OR     X34	; 料盘到位光纤，上料，产品盘2
ANB
DMOV   HSD0 D10
RST    M225
LD     SM0
DSUB   HSD0 D10 D14	; 上顶圈数计数
LD     M224
LD     X10102	; 料盘到位光纤，上料，产品盘
AND    X34	; 料盘到位光纤，上料，产品盘2
DOR>   D14 K15000	; 上顶圈数计数
ORI    X15	; 上料1模组上光电开关【常闭】
ANB
RST    S8	; S8防止料盘斜，上顶动作
RST    M225
DMOV   K0 D14	; 上顶圈数计数
RST    M0	; 启动上料轴1
STOP   Y0 K1	; 上料1电机脉冲
RST    M224
LD     M224
AND    M100	; 公共暂停
SET    M223
RST    M0	; 启动上料轴1
STOP   Y0 K1	; 上料1电机脉冲
RST    M224
STLE
STL    S219	; S219上料轴先下降10mm
LDP    S219	; S219上料轴先下降10mm
SET    M310
DMOV   HSD0 D200	; 记录轴1当前位置

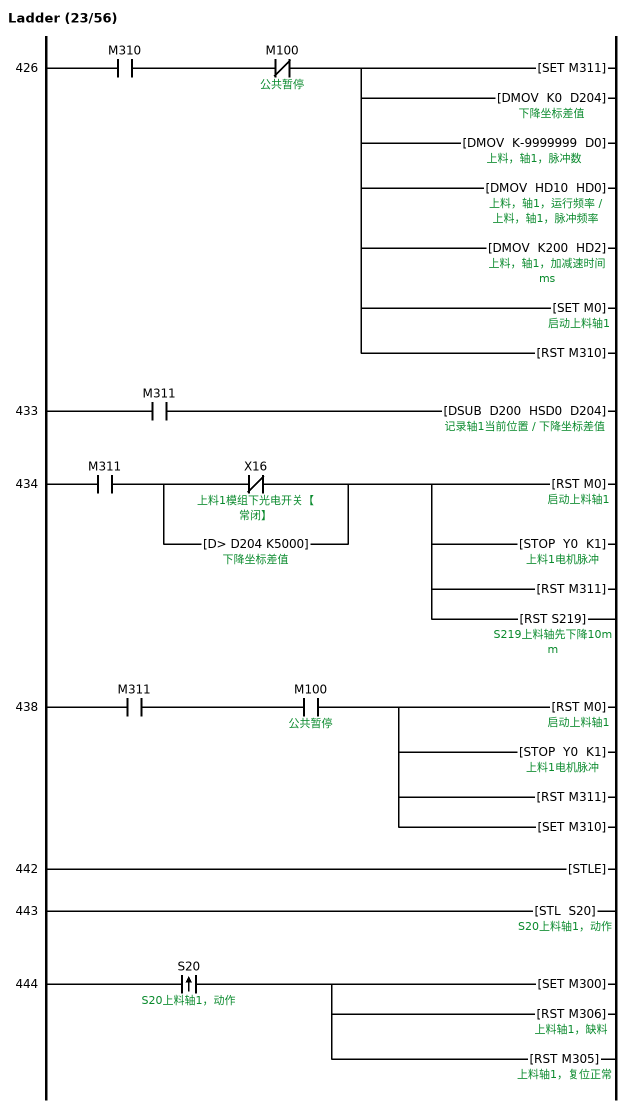
LD     M310
ANI    M100	; 公共暂停
SET    M311
DMOV   K0 D204	; 下降坐标差值
DMOV   K-9999999 D0	; 上料，轴1，脉冲数
DMOV   HD10 HD0	; 上料，轴1，运行频率 / 上料，轴1，脉冲频率
DMOV   K200 HD2	; 上料，轴1，加减速时间ms
SET    M0	; 启动上料轴1
RST    M310
LD     M311
DSUB   D200 HSD0 D204	; 记录轴1当前位置 / 下降坐标差值
LD     M311
LDI    X16	; 上料1模组下光电开关【常闭】
DOR>   D204 K5000	; 下降坐标差值
ANB
RST    M0	; 启动上料轴1
STOP   Y0 K1	; 上料1电机脉冲
RST    M311
RST    S219	; S219上料轴先下降10mm
LD     M311
AND    M100	; 公共暂停
RST    M0	; 启动上料轴1
STOP   Y0 K1	; 上料1电机脉冲
RST    M311
SET    M310
STLE
STL    S20	; S20上料轴1，动作
LDP    S20	; S20上料轴1，动作
SET    M300
RST    M306	; 上料轴1，缺料
RST    M305	; 上料轴1，复位正常

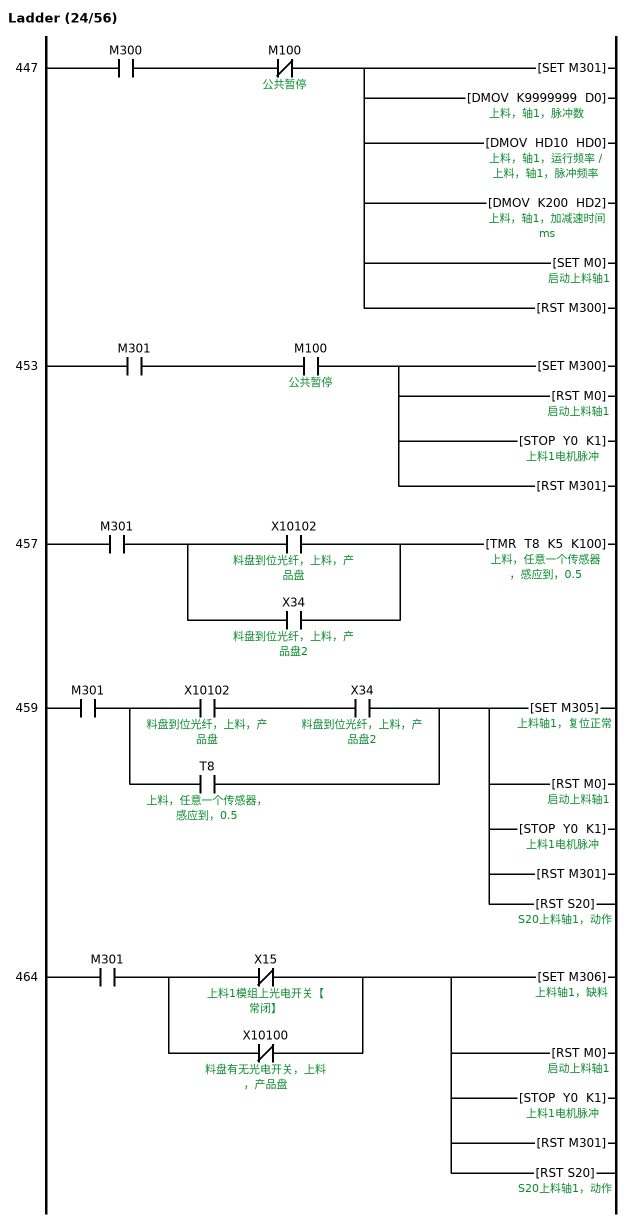
LD     M300
ANI    M100	; 公共暂停
SET    M301
DMOV   K9999999 D0	; 上料，轴1，脉冲数
DMOV   HD10 HD0	; 上料，轴1，运行频率 / 上料，轴1，脉冲频率
DMOV   K200 HD2	; 上料，轴1，加减速时间ms
SET    M0	; 启动上料轴1
RST    M300
LD     M301
AND    M100	; 公共暂停
SET    M300
RST    M0	; 启动上料轴1
STOP   Y0 K1	; 上料1电机脉冲
RST    M301
LD     M301
LD     X10102	; 料盘到位光纤，上料，产品盘
OR     X34	; 料盘到位光纤，上料，产品盘2
ANB
TMR    T8 K5 K100	; 上料，任意一个传感器，感应到，0.5
LD     M301
LD     X10102	; 料盘到位光纤，上料，产品盘
AND    X34	; 料盘到位光纤，上料，产品盘2
OR     T8	; 上料，任意一个传感器，感应到，0.5
ANB
SET    M305	; 上料轴1，复位正常
RST    M0	; 启动上料轴1
STOP   Y0 K1	; 上料1电机脉冲
RST    M301
RST    S20	; S20上料轴1，动作
LD     M301
LDI    X15	; 上料1模组上光电开关【常闭】
ORI    X10100	; 料盘有无光电开关，上料，产品盘
ANB
SET    M306	; 上料轴1，缺料
RST    M0	; 启动上料轴1
STOP   Y0 K1	; 上料1电机脉冲
RST    M301
RST    S20	; S20上料轴1，动作

